TYPE "UDT_ZC_SIVE_MEMBRANA_CARE"
VERSION : 0.1
   STRUCT
      FechaHora { S7_SetPoint := 'False'} : "UDT_ZC_FECHA";   // Fecha y hora del registro
      TiempoMembrana : UDInt;   // Tiempo de la membrana
      Tecnico : String[20];   // Tecnico a cargo
   END_STRUCT;

END_TYPE

